Fanuc KAREL source: ko00092.KL

-- PROVISIONAL review KL for V1013-1; original PC SHA256 a27562421798afd71af29620257d8728fe9c9c3a36e81b65f0563d15f56f31af
-- Incomplete behavior may be omitted. Consult companion uncertainty JSON. Do not deploy.
PROGRAM KO00092
%NOLOCKGROUP
BEGIN
  -- UNRESOLVED_PC offsets 5-12; opcodes 9D,23
  -- UNRESOLVED_PC offsets 17-69; opcodes 27,27,49,7E,AD,27,49,7E,AD,22,31,7E,4A
  -- UNRESOLVED_PC offsets 74-78; opcodes 7F
END KO00092
